// TIA Portal V15.1 export
// export: Created 2024-05-17T05:38:25.9667863Z, ExportSetting WithDefaults, DisplayName Totally Integrated Automation Portal, DisplayVersion V15.1 Update 5, DisplayName TIA Portal Openness, DisplayVersion V15.1 Update 5, DisplayName SINAMICS Startdrive Advanced, DisplayVersion V15.1, DisplayName G130, G150, S120, S150, SINAMICS MV, S210, DisplayVersion V15.1, DisplayName G110M, G120, G120C, G120D, G120P, DisplayVersion V15.1, DisplayName STEP 7 Professional, DisplayVersion V15.1 Update 5, DisplayName STEP 7 Safety, DisplayVersion V15.1, DisplayName WinCC Professional, DisplayVersion V15.1 Update 5, DisplayName SIMATIC Visualization Architect, DisplayVersion V15.1
FUNCTION "LWordToBit" : Void   // FC1001, FBD
TITLE = LWordToBit
{ S7_Optimized_Access := 'FALSE' }
AUTHOR : VCC
FAMILY : Control
NAME : Word2Bit
VERSION : 1.0
// ================================================================================
// Moves One Word to 16 bits 
// ================================================================================
// stored: AutoNumber false, IsIECCheckEnabled false, SetENOAutomatically False, UDAEnableTagReadback false
   VAR_INPUT
      I_Word : Word;   // Input Word
   END_VAR
   VAR_OUTPUT
      O_0 : Bool;   // Output 0
      O_1 : Bool;   // Output 1
      O_2 : Bool;   // Output 2
      O_3 : Bool;   // Output 3
      O_4 : Bool;   // Output 4
      O_5 : Bool;   // Output 5
      O_6 : Bool;   // Output 6
      O_7 : Bool;   // Output 7
      O_8 : Bool;   // Output 8
      O_9 : Bool;   // Output 9
      O_10 : Bool;   // Output 10
      O_11 : Bool;   // Output 11
      O_12 : Bool;   // Output 12
      O_13 : Bool;   // Output 13
      O_14 : Bool;   // Output 14
      O_15 : Bool;   // Output 15
   END_VAR
BEGIN

REGION Network 1: **** 8 - Outputs ****
   // Copy bit 0 from Word to output
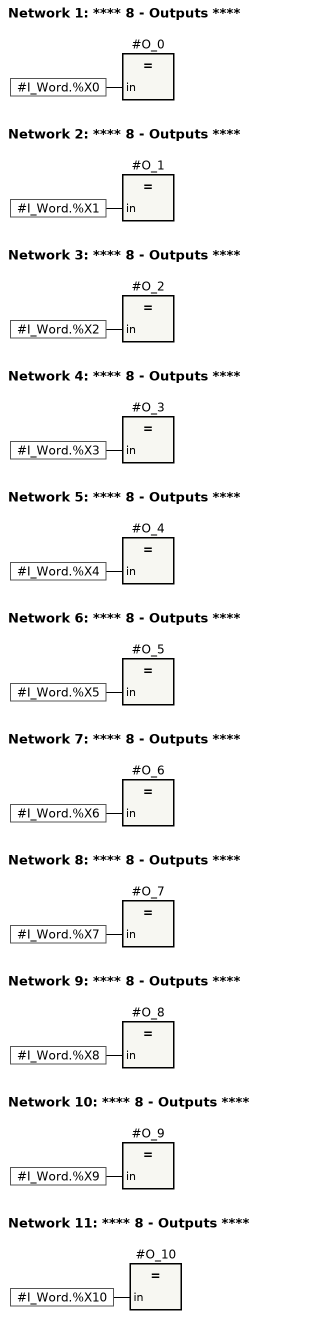
   #O_0 := #I_Word.%X0;
END_REGION

REGION Network 2: **** 8 - Outputs ****
   // Copy bit 1 from Word to output
   #O_1 := #I_Word.%X1;
END_REGION

REGION Network 3: **** 8 - Outputs ****
   // Copy bit 2 from Word to output
   #O_2 := #I_Word.%X2;
END_REGION

REGION Network 4: **** 8 - Outputs ****
   // Copy bit 3 from Word to output
   #O_3 := #I_Word.%X3;
END_REGION

REGION Network 5: **** 8 - Outputs ****
   // Copy bit 4 from Word to output
   #O_4 := #I_Word.%X4;
END_REGION

REGION Network 6: **** 8 - Outputs ****
   // Copy bit 5 from Word to output
   #O_5 := #I_Word.%X5;
END_REGION

REGION Network 7: **** 8 - Outputs ****
   // Copy bit 6 from Word to output
   #O_6 := #I_Word.%X6;
END_REGION

REGION Network 8: **** 8 - Outputs ****
   // Copy bit 7 from Word to output
   #O_7 := #I_Word.%X7;
END_REGION

REGION Network 9: **** 8 - Outputs ****
   // Copy bit 8 from Word to output
   #O_8 := #I_Word.%X8;
END_REGION

REGION Network 10: **** 8 - Outputs ****
   // Copy bit 9 from Word to output
   #O_9 := #I_Word.%X9;
END_REGION

REGION Network 11: **** 8 - Outputs ****
   // Copy bit 10 from Word to output
   #O_10 := #I_Word.%X10;
END_REGION

REGION Network 12: **** 8 - Outputs ****
   // Copy bit 11 from Word to output
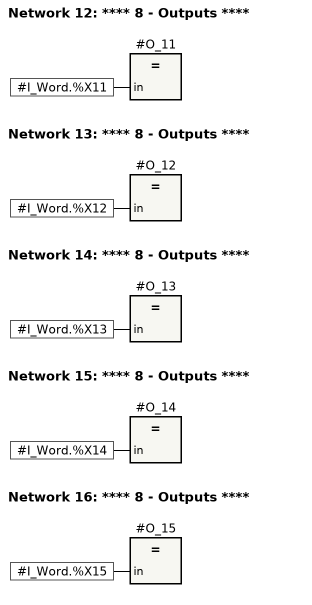
   #O_11 := #I_Word.%X11;
END_REGION

REGION Network 13: **** 8 - Outputs ****
   // Copy bit 12 from Word to output
   #O_12 := #I_Word.%X12;
END_REGION

REGION Network 14: **** 8 - Outputs ****
   // Copy bit 13 from Word to output
   #O_13 := #I_Word.%X13;
END_REGION

REGION Network 15: **** 8 - Outputs ****
   // Copy bit 14 from Word to output
   #O_14 := #I_Word.%X14;
END_REGION

REGION Network 16: **** 8 - Outputs ****
   // Copy bit 15 from Word to output
   #O_15 := #I_Word.%X15;
END_REGION
END_FUNCTION
